{attribute 'linkalways'} 
{attribute 'no_explicit_call' := 'This FB is a CLASS and must be accessed using methods or properties'}
{attribute 'enable_dynamic_creation'}
FUNCTION_BLOCK Node_F_VN_SetAt_TcVnVector3_UINT EXTENDS VisionNode
VAR
    aElement : _TcVnVector3_UINT;
    ipContainer : _ITcVnContainer;
    nIndex : _ULINT(0);
    hrPrev : _HRESULT(S_OK);
    hresult : _HRESULT(S_OK);
END_VAR

METHOD PUBLIC  Clone : I_Node
VAR
	pNode : POINTER TO Node_F_VN_SetAt_TcVnVector3_UINT;
END_VAR
pNode := __NEW(Node_F_VN_SetAt_TcVnVector3_UINT);
Clone := pNode^;
END_METHOD

METHOD FB_init : BOOL
VAR_INPUT
	bInitRetains : BOOL; // if TRUE, the retain variables are initialized (warm start / cold start)
	bInCopyCode : BOOL;  // if TRUE, the instance afterwards gets moved into the copy code (online change)
END_VAR
AddInput('aElement', aElement);
AddInput('ipContainer', ipContainer);
AddInput('nIndex', nIndex);
AddInput('hrPrev', hrPrev);
AddOutput('ipContainer', ipContainer);
AddOutput('hresult',hresult);
END_METHOD

METHOD PROTECTED OnExecute : HRESULT
hresult.Value := F_VN_SetAt_TcVnVector3_UINT(
    aElement := aElement.Value,
    ipContainer := ipContainer.Value,
    nIndex := nIndex.Value,
    hrPrev:= hrPrev.Value);
END_METHOD

METHOD PUBLIC PreExecutionCheck
VAR_INPUT
	Check : I_PreExecutionChecks;
END_VAR
Check.IsTrue(ipContainer.IsValid, 'ipContainer must be a valid container');
END_METHOD

END_FUNCTION_BLOCK

(* stored: Version 1.1.0.1, ProductVersion 3.1.4024.13
   POU Node_F_VN_SetAt_TcVnVector3_UINT: Id {49b5e89b-7ee5-411b-bc6c-6241bfb44171}, SpecialFunc None
   Folder Constructor: Id {5ca2f5e1-226e-43c5-9f25-432615789352}
   Method Clone: Id {bd0f5443-db75-4cb5-a1e7-08edcb00a952}
   Method FB_init: Id {152a423d-398a-4f10-9101-8b5838a41fb3}
   Method OnExecute: Id {b06fcec0-0b49-4897-996a-6df043cecddc}
   Method PreExecutionCheck: Id {28bdb9e3-4c0c-4a89-b90d-46732362528b} *)
